FUNCTION_BLOCK Conveyor1Check (* Template for a Basic Function Block Type *)
  (* Standard: 61499-2 *)
  (* Version 1.0, 2021-07-29, Tuojian Lyu *)
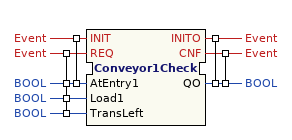
  EVENT_INPUT
    INIT WITH AtEntry1; (* Initialization Request *)
    REQ WITH AtEntry1, Load1, TransLeft; (* Normal Execution Request *)
  END_EVENT
  EVENT_OUTPUT
    INITO WITH QO; (* Initialization Confirm *)
    CNF WITH QO; (* Execution Confirmation *)
  END_EVENT
  VAR_INPUT
    AtEntry1 : BOOL; (* Input event qualifier *)
    Load1 : BOOL;
    TransLeft : BOOL;
  END_VAR
  VAR_OUTPUT
    QO : BOOL; (* Output event qualifier *)
  END_VAR
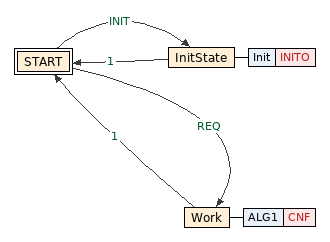
  EC_STATES
    START; (* Initial State *)
    InitState : Init -> INITO;
    Work : ALG1 -> CNF;
  END_STATES
  EC_TRANSITIONS
    START TO InitState := INIT;
    InitState TO START := 1;
    START TO Work := REQ;
    Work TO START := 1;
  END_TRANSITIONS
  ALGORITHM Init IN ST:
QO := TRUE;
  END_ALGORITHM
  ALGORITHM ALG1 IN ST:
IF (TRUE = TransLeft) THEN
QO := FALSE;
ELSE
QO := TRUE;
END_IF;
  END_ALGORITHM
END_FUNCTION_BLOCK
